FUNCTION_BLOCK FB_PrintOverview
VAR_INPUT
  fResSubPx     : LREAL;   // Subpixel pulse resolution
END_VAR

VAR
  // helper
  bInit   : BOOL;
  nCtr    : UDINT;
  nNum    : UDINT;
  
  // config
  _pCTM   : POINTER TO FB_CTManagerDts;
  _fPrintResolution : LREAL;      // [dpi]
  _fSubPixelResolution : LREAL;   // sub pixel resolution [x]
  
  // Container view list
  iCT     : I_CT;
  aCTV    : ARRAY[1..iCPr_MAX_CONTAINER] OF FB_ContainerView;
  // Worker view list
  iWorker : I_Worker;
  
  // motion and position
  bMovingInd : BOOL;
  fSpeed  : LREAL;
  fbBlink : FB_BLINK;
  t : TIME;
  
  // time
  sCurrentDateTime : STRING;
END_VAR

VAR CONSTANT
  nC_MAX_WORKER_VIEWS : UINT := 10;
END_VAR

IF NOT checkConfig() THEN RETURN; END_IF    // check config

// -- current time ---------------------------
sCurrentDateTime := F_TimeGetDateTime();

METHOD checkConfig : BOOL
VAR_INPUT
END_VAR
VAR_INST
  _fX_m, _fY_m   : LREAL;
  _nX_px, _nY_px : DINT; 
END_VAR
VAR
  bOK : BOOL;
END_VAR
IF NOT bInit THEN RETURN; END_IF

checkConfig := TRUE;
END_METHOD

METHOD init : BOOL
VAR_INPUT
  pCTM                : POINTER TO FB_CTManager;
  fSubPixelResolution : LREAL;
END_VAR
IF pCTM = 0 THEN RETURN; END_IF

_pCTM := pCTM;

bInit := TRUE;
END_METHOD

END_FUNCTION_BLOCK

(* stored: Version 1.1.0.1, ProductVersion 3.1.4024.9
   POU FB_PrintOverview: Id {57a6df33-c5fc-4b78-b796-858abcecd4f4}, SpecialFunc None
   Method checkConfig: Id {edfe75ad-63c4-4ec1-9d31-8e206962e7b0}
   Method init: Id {bd002f50-5fd9-48d9-b817-a794ac96eb55} *)
